FUNCTION TryConvert_ULINT_TO_SINT : BOOL
VAR_INPUT
	in : ULINT;
	out : REFERENCE TO SINT;
END_VAR

IF in > DatatypeLimits.MAX_VALUE_OF_ULINT_WHICH_CAN_BE_HELD_IN_A_SINT THEN
	RETURN;
END_IF

out := ULINT_TO_SINT(in);
TryConvert_ULINT_TO_SINT := TRUE;

END_FUNCTION

(* stored: Version 1.1.0.1, ProductVersion 3.1.4024.12
   POU TryConvert_ULINT_TO_SINT: Id {8076b988-f20f-43b0-a9e3-1769287ef806}, SpecialFunc None *)
